(* IEC 61131-3 sources: Industry-PLC-LLM/data/PLCBEAD_repo/PLCBEAD_PLCEmbed-main/PLC-BEAD/Source/GEB/MUX_2, 1 file *)

(* ---- MUX_2.ST ---- *)
FUNCTION MUX_2:BOOL

	VAR_INPUT
		D0 :	BOOL;
		D1 :	BOOL;
		A0 :	BOOL;
	END_VAR

	MUX_2 := SEL(A0, D0, D1);

END_FUNCTION

PROGRAM program0
	VAR
		D0 :	BOOL;
		D1 :	BOOL;
		A0 :	BOOL;
		OUT : BOOL;
	END_VAR

	OUT := MUX_2(D0, D1, A0);

END_PROGRAM
